// TIA Portal V17 export
// export: Created 2025-06-26T06:49:11.315232Z, ExportSetting WithDefaults, DisplayName Totally Integrated Automation Portal, DisplayVersion V17 Update 8, DisplayName TIA Portal Openness, DisplayVersion V17 Update 8, DisplayName TIA Portal Version Control Interface, DisplayVersion V17, DisplayName STEP 7 Professional, DisplayVersion V17 Update 8, DisplayName STEP 7 Safety, DisplayVersion V17 Update 6, DisplayName WinCC Advanced, DisplayVersion V17 Update 8
FUNCTION_BLOCK "Simulation"   // FB63, FBD
TITLE = Simulation of process values
{ S7_Optimized_Access := 'TRUE' }
AUTHOR : Heaten
VERSION : 0.1
// Simulate process values
// stored: AutoNumber true, IsIECCheckEnabled false, IsRetainMemResEnabled false, MemoryReserve 0, SetENOAutomatically false, UDAEnableTagReadback false
   VAR
      OilSump { S7_SetPoint := 'True'} : "fbButterworthLPF1";
      CPCPump { ExternalAccessible := 'False'; ExternalVisible := 'False'; ExternalWritable := 'False'; S7_SetPoint := 'True'} : "fbCPCPumpSim";
      HeatSource { S7_SetPoint := 'True'} : "fbButterworthLPF1";
   END_VAR
   VAR RETAIN
      fHeatSourceGain { S7_SetPoint := 'True'} : Real := 1.2;   // Conversion factor, % valve opening to HX temperature
   END_VAR
   VAR_TEMP
      fSumpHeatingTarget : Real;
      fOilSumpTemp : Real;
      fCPCDischarge : Real;
      fHeatSourceTarget : Real;
      fHeatSourceSimulated : Real;
   END_VAR
   VAR_TEMP   // added for the SCL form of the ladder/FBD networks
      _w1 : Bool;
   END_VAR
BEGIN

REGION Network 1 (SCL): Block comments
   // Don't put as comments under Block Title as this automatically appears in the weirdest places
   // A collection of hacks to provide feedback from the missing physical processes
END_REGION

REGION Network 2 (SCL): Simulation HBL-SC-10
   IF "DB_Alarms"."1110_HBL_SC_10_CommError".sState.bActive = TRUE THEN
       "DB_InverterDrives".HBL_SC_10.Stat.bOnline := TRUE;
       "DB_InverterDrives".HBL_SC_10.Stat.bReady := "DB_InverterDrives".HBL_SC_10.Cmd.bReady OR "DB_InverterDrives".HBL_SC_10.Cmd.bRun;
       "DB_InverterDrives".HBL_SC_10.Stat.bRemote := TRUE;
       "DB_InverterDrives".HBL_SC_10.Stat.bRun := "DB_InverterDrives".HBL_SC_10.Cmd.bRun;
       "DB_InverterDrives".HBL_SC_10.Stat.Speed.Eng.bError := FALSE;
       "DB_InverterDrives".HBL_SC_10.Stat.Speed.Eng.fValue :="DB_InverterDrives".HBL_SC_10.Cmd.Speed.Eng.fValue;
       "DB_InverterDrives".HBL_SC_10.Stat.Torque.Eng.bError := FALSE;
       "DB_InverterDrives".HBL_SC_10.Stat.Torque.Eng.fValue := "DB_InverterDrives".HBL_SC_10.Cmd.Torque.Eng.fValue;
       "DB_InverterDrives".HBL_SC_10.Stat.Power.Eng.bError := FALSE;
       "DB_InverterDrives".HBL_SC_10.Stat.Power.Eng.fValue := 355.0 * "DB_InverterDrives".HBL_SC_10.Stat.Speed.Eng.fValue/1500.0;
   END_IF;
END_REGION

REGION Network 3 (SCL): Simulation for oil gallery pressure
   // Just a rough hack to get some representative pressures
   // Oil pressure is always the sum of the two pumps. The primer pump will drop out above a certain oil pressure and come back on
   // We let the regulator decide for us and just do the sum
   // Primer pump: 100kPa at 5000rpm = 0.02 kPa/rpm (0.021747 to make it look more "random")
   // Main pump: 0.250 kPa/rpm to be above the minimum of 0.167 kPa/rpm to avoid warnings (0.257 to make it look more "random")
   // Filter deltaP = 20kPa
   "fcCalcAssign"(fValue := "DB_InverterDrives".HBL_SC_02.Stat.Speed.Eng.fValue * 0.021747 + "DB_InverterDrives".HBL_SC_10.Stat.Speed.Eng.fValue * 0.257,
                  sTag := "DB_AI".HBL_PT_960.Eng);
   "DB_AI".HBL_PT_961.Eng.bCheckLimits := TRUE;   // Limit to min & max
   "fcCalcAssign"(fValue := "DB_AI".HBL_PT_960.Eng.fValue - 20.0, sTag := "DB_AI".HBL_PT_961.Eng);
END_REGION

REGION Network 4: Simulation for Oil Sump Temperature
   // Thermal time constant: estimate 30 minutes to go from ambient to 45C
   // 5 tau = 30 minutes, or tau = 360 sec, or fc = 1/(2*pi*tau) = 0.00044210Hz (0.44mHz)
   // Go to 45C on Group 1 heaters, go to 82C on Group 1 + 2 heaters
   // When cooling, go towards the container air temperature
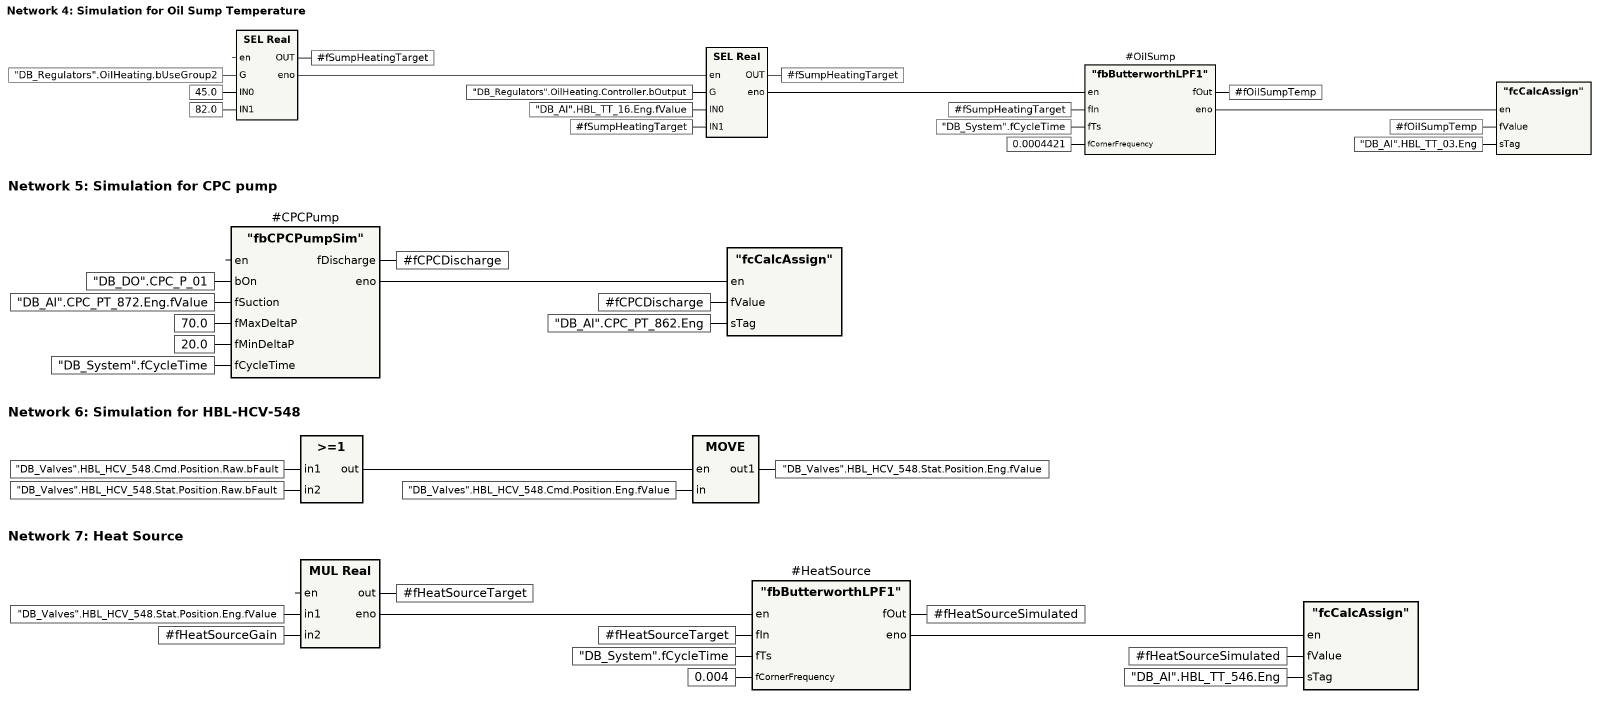
   // ENO of a box is taken as its EN; it also drops when the box reports an error
   #fSumpHeatingTarget := SEL(G := "DB_Regulators".OilHeating.bUseGroup2, IN0 := 45.0, IN1 := 82.0);
   #fSumpHeatingTarget := SEL(G := "DB_Regulators".OilHeating.Controller.bOutput, IN0 := "DB_AI".HBL_TT_16.Eng.fValue, IN1 := #fSumpHeatingTarget);
   #OilSump(fIn := #fSumpHeatingTarget,   // "fbButterworthLPF1"
            fTs := "DB_System".fCycleTime,
            fCornerFrequency := 0.0004421,
            fOut => #fOilSumpTemp,
            ENO => #_w1);
   IF #_w1 THEN "fcCalcAssign"(fValue := #fOilSumpTemp, sTag := "DB_AI".HBL_TT_03.Eng); END_IF;
END_REGION

REGION Network 5: Simulation for CPC pump
   #CPCPump(bOn := "DB_DO".CPC_P_01,   // "fbCPCPumpSim"
            fSuction := "DB_AI".CPC_PT_872.Eng.fValue,
            fMaxDeltaP := 70.0,
            fMinDeltaP := 20.0,
            fCycleTime := "DB_System".fCycleTime,
            fDischarge => #fCPCDischarge,
            ENO => #_w1);
   IF #_w1 THEN "fcCalcAssign"(fValue := #fCPCDischarge, sTag := "DB_AI".CPC_PT_862.Eng); END_IF;
END_REGION

REGION Network 6: Simulation for HBL-HCV-548
   // Only overwrite if the valve is not simulated electrically
   IF "DB_Valves".HBL_HCV_548.Cmd.Position.Raw.bFault OR "DB_Valves".HBL_HCV_548.Stat.Position.Raw.bFault THEN
       "DB_Valves".HBL_HCV_548.Stat.Position.Eng.fValue := "DB_Valves".HBL_HCV_548.Cmd.Position.Eng.fValue;
   END_IF;
END_REGION

REGION Network 7: Heat Source
   // Simulate heat source suction temperature
   #fHeatSourceTarget := "DB_Valves".HBL_HCV_548.Stat.Position.Eng.fValue * #fHeatSourceGain;
   #HeatSource(fIn := #fHeatSourceTarget,   // "fbButterworthLPF1"
               fTs := "DB_System".fCycleTime,
               fCornerFrequency := 0.004,
               fOut => #fHeatSourceSimulated,
               ENO => #_w1);
   IF #_w1 THEN "fcCalcAssign"(fValue := #fHeatSourceSimulated, sTag := "DB_AI".HBL_TT_546.Eng); END_IF;
END_REGION
END_FUNCTION_BLOCK
